// TIA Portal project "zbiorniki" (V15)

(* hardware
DEVICE "S7-1200 station_1"  S7-1200 Station
   slot 0: "Rack_0"  S7-1200 Rack  Rack  V1.0
   slot 1: "PLC_1"  CPU 1214C DC/DC/DC  6ES7 214-1AG40-0XB0  V4.2
      slot 3: "AQ 1x12BIT_1"  AQ1 signal board  6ES7 232-4HA30-0XB0  V1.0
   slot 101: "CM 1243-5"  CM 1243-5  6GK7 243-5DX30-0XE0  V1.3
   slot 102: "CM 1241 (RS485)_1"  CM 1241 (RS485)  6ES7 241-1CH30-0XB0  V1.0
*)

// ===== PLC "PLC_1"  CPU 1214C DC/DC/DC =====

VAR_GLOBAL   // PLC tag table "Default tag table"
   "czujnikDol1" AT %I0.0 : Bool;
   "czujnikGora1" AT %I0.1 : Bool;
   "Tag_2" AT %M0.0 : Bool;
   "Tag_3" AT %M0.1 : Bool;
   "Tag_4" AT %M0.2 : Bool;
   "Tag_5" AT %M2.0 : Bool;
   "poziomWodyZbiornik2" AT %MW1 : Int;
   "Tag_6" AT %IW64 : Int;
   "analog" AT %MD100 : Real;
   "skalowana" AT %MW104 : Int;
   "czujnikD2" AT %I0.2 : Bool;
   "czujnikG2" AT %I0.3 : Bool;
   "Tag_9" AT %M50.0 : Bool;
   "Tag_10" AT %M50.1 : Bool;
   "Tag_11" AT %M50.2 : Bool;
END_VAR

DATA_BLOCK "zbiornik_DB1"   // DB1
{ S7_Optimized_Access := 'TRUE' }
VERSION : 0.1
// stored: InstanceOfName zbiornik
"zbiornik"
BEGIN
   poziomCieczy := 1000;
END_DATA_BLOCK

DATA_BLOCK "pompa_DB1"   // DB2
{ S7_Optimized_Access := 'TRUE' }
VERSION : 0.1
// stored: InstanceOfName pompa
"pompa"
BEGIN
END_DATA_BLOCK

DATA_BLOCK "zbiornik_DB2"   // DB3
{ S7_Optimized_Access := 'TRUE' }
VERSION : 0.1
// stored: InstanceOfName zbiornik
"zbiornik"
BEGIN
   poziomCieczy := 500;
END_DATA_BLOCK

DATA_BLOCK "pompa_DB2"   // DB4
{ S7_Optimized_Access := 'TRUE' }
VERSION : 0.1
// stored: InstanceOfName pompa
"pompa"
BEGIN
END_DATA_BLOCK

FUNCTION_BLOCK "zbiornik"   // FB1, LAD
{ S7_Optimized_Access := 'TRUE' }
VERSION : 0.1
   VAR_INPUT
      czujnikD : Bool;
      czujnikG : Bool;
   END_VAR
   VAR_OUTPUT
      zbiornikPusty : Bool;
      zbiornikPolowa : Bool;
      zbiornikPelen : Bool;
   END_VAR
   VAR_IN_OUT
      poziomCieczy : Int;
   END_VAR
BEGIN

REGION Network 1: zbiornik pusty
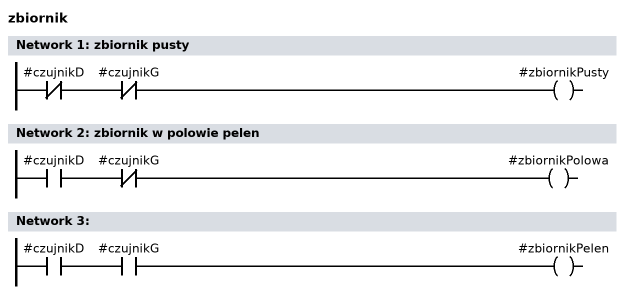
   RUNG wire#powerrail
      I_Contact( #czujnikD )
      I_Contact( #czujnikG )
      Coil( #zbiornikPusty )
   END_RUNG
   // the same network as SCL:
   #zbiornikPusty := NOT #czujnikD AND NOT #czujnikG;
END_REGION

REGION Network 2: zbiornik w polowie pelen
   RUNG wire#powerrail
      Contact( #czujnikD )
      I_Contact( #czujnikG )
      Coil( #zbiornikPolowa )
   END_RUNG
   // the same network as SCL:
   #zbiornikPolowa := #czujnikD AND NOT #czujnikG;
END_REGION

REGION Network 3
   RUNG wire#powerrail
      Contact( #czujnikD )
      Contact( #czujnikG )
      Coil( #zbiornikPelen )
   END_RUNG
   // the same network as SCL:
   #zbiornikPelen := #czujnikD AND #czujnikG;
END_REGION
END_FUNCTION_BLOCK

FUNCTION_BLOCK "pompa"   // FB2, LAD
{ S7_Optimized_Access := 'TRUE' }
VERSION : 0.1
   VAR_INPUT
      poziomCieczy : Int;
      poziomGorny : Bool;
      wysokosc : Int;
   END_VAR
   VAR_IN_OUT
      pracaPompyZb1 : Bool;
   END_VAR
BEGIN

REGION Network 1: praca pompy
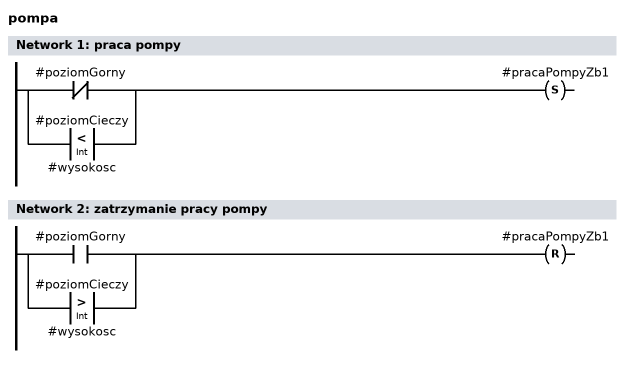
   RUNG wire#powerrail
      I_Contact( #poziomGorny )
      wire#w1
      S_Coil( #pracaPompyZb1 )
   END_RUNG
   RUNG wire#powerrail
      { S7_Templates := "SrcType := Int" } LT_Contact(in1 := #poziomCieczy, in2 := #wysokosc)
   END_RUNG wire#w1
   // the same network as SCL:
   IF NOT #poziomGorny OR (#poziomCieczy < #wysokosc) THEN #pracaPompyZb1 := TRUE; END_IF;
END_REGION

REGION Network 2: zatrzymanie pracy pompy
   RUNG wire#powerrail
      Contact( #poziomGorny )
      wire#w1
      R_Coil( #pracaPompyZb1 )
   END_RUNG
   RUNG wire#powerrail
      { S7_Templates := "SrcType := Int" } GT_Contact(in1 := #poziomCieczy, in2 := #wysokosc)
   END_RUNG wire#w1
   // the same network as SCL:
   IF #poziomGorny OR (#poziomCieczy > #wysokosc) THEN #pracaPompyZb1 := FALSE; END_IF;
END_REGION
END_FUNCTION_BLOCK

FUNCTION "przeplyw" : Void   // FC1, LAD
{ S7_Optimized_Access := 'TRUE' }
VERSION : 0.1
   VAR_INPUT
      zbiornik1 : Int;
      zmiana : Int;
      zbiornik2 : Int;
   END_VAR
   VAR_OUTPUT
      roznicaZbiornk1 : Int;
      roznicaZbiornik2 : Int;
   END_VAR
BEGIN

REGION Network 1: poziom wody w zbiorniku 2
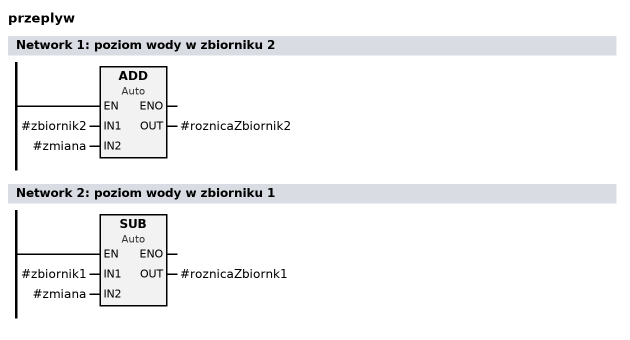
   RUNG wire#powerrail
      Add(in1 := #zbiornik2, in2 := #zmiana, out => #roznicaZbiornik2)
   END_RUNG
   // the same network as SCL:
   #roznicaZbiornik2 := #zbiornik2 + #zmiana;
END_REGION

REGION Network 2: poziom wody w zbiorniku 1
   RUNG wire#powerrail
      Sub(in1 := #zbiornik1, in2 := #zmiana, out => #roznicaZbiornk1)
   END_RUNG
   // the same network as SCL:
   #roznicaZbiornk1 := #zbiornik1 - #zmiana;
END_REGION
END_FUNCTION

ORGANIZATION_BLOCK "Main"   // OB1, LAD, ProgramCycle
TITLE = "Main Program Sweep (Cycle)"
{ S7_Optimized_Access := 'TRUE' }
VERSION : 0.1
   VAR_INPUT
      Initial_Call : Bool;   // Initial call of this OB
      Remanence : Bool;   // =True, if remanent data are available
   END_VAR
BEGIN

REGION Network 1: odczyt analogowy (poziom cieczy)
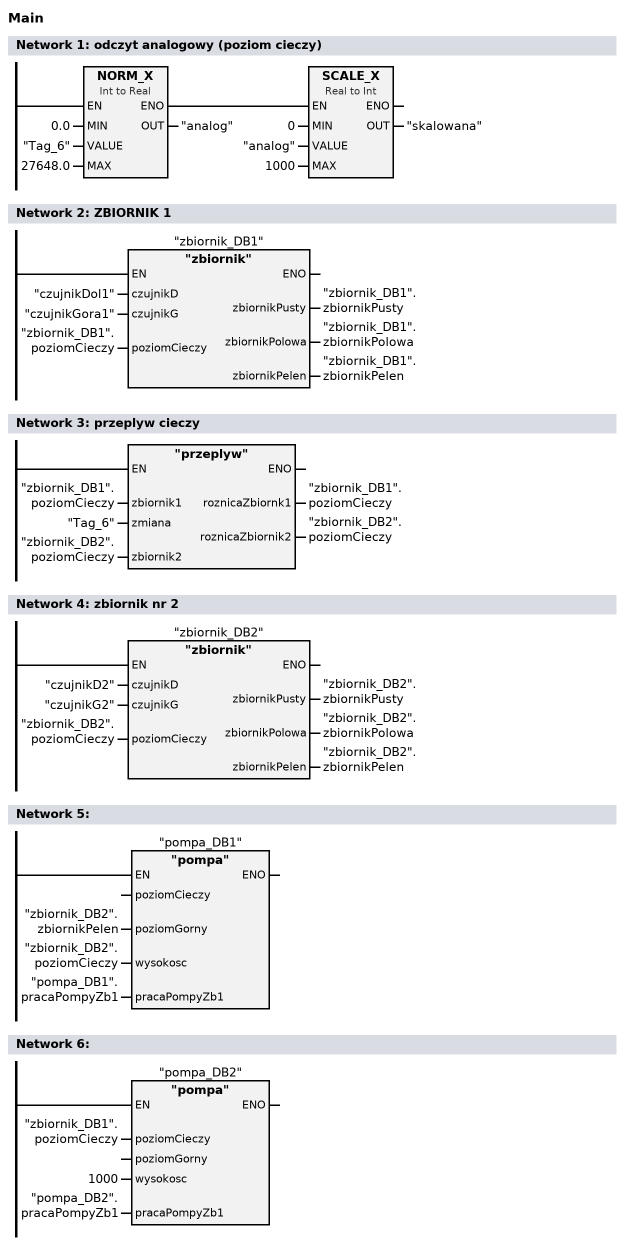
   RUNG wire#powerrail
      { S7_Templates := "[SrcType := Int, DestType := Real]" } Normalize(min := 0.0, value := "Tag_6", max := 27648.0, out => "analog")
      { S7_Templates := "[SrcType := Real, DestType := Int]" } Scale(min := 0, value := "analog", max := 1000, out => "skalowana")
   END_RUNG
   // the same network as SCL:
   "analog" := NORM_X(MIN := 0.0, VALUE := "Tag_6", MAX := 27648.0);
   "skalowana" := SCALE_X(MIN := 0, VALUE := "analog", MAX := 1000);
END_REGION

REGION Network 2: ZBIORNIK 1
   RUNG wire#powerrail
      "zbiornik_DB1"(czujnikD := "czujnikDol1", czujnikG := "czujnikGora1", poziomCieczy := "zbiornik_DB1".poziomCieczy, zbiornikPusty => "zbiornik_DB1".zbiornikPusty, zbiornikPolowa => "zbiornik_DB1".zbiornikPolowa, zbiornikPelen => "zbiornik_DB1".zbiornikPelen)
   END_RUNG
   // the same network as SCL:
   "zbiornik_DB1"(czujnikD := "czujnikDol1",   // "zbiornik"
                  czujnikG := "czujnikGora1",
                  poziomCieczy := "zbiornik_DB1".poziomCieczy,
                  zbiornikPusty => "zbiornik_DB1".zbiornikPusty,
                  zbiornikPolowa => "zbiornik_DB1".zbiornikPolowa,
                  zbiornikPelen => "zbiornik_DB1".zbiornikPelen);
END_REGION

REGION Network 3: przeplyw cieczy
   RUNG wire#powerrail
      "przeplyw"(zbiornik1 := "zbiornik_DB1".poziomCieczy, zmiana := "Tag_6", zbiornik2 := "zbiornik_DB2".poziomCieczy, roznicaZbiornk1 => "zbiornik_DB1".poziomCieczy, roznicaZbiornik2 => "zbiornik_DB2".poziomCieczy)
   END_RUNG
   // the same network as SCL:
   "przeplyw"(zbiornik1 := "zbiornik_DB1".poziomCieczy,
              zmiana := "Tag_6",
              zbiornik2 := "zbiornik_DB2".poziomCieczy,
              roznicaZbiornk1 => "zbiornik_DB1".poziomCieczy,
              roznicaZbiornik2 => "zbiornik_DB2".poziomCieczy);
END_REGION

REGION Network 4: zbiornik nr 2
   RUNG wire#powerrail
      "zbiornik_DB2"(czujnikD := "czujnikD2", czujnikG := "czujnikG2", poziomCieczy := "zbiornik_DB2".poziomCieczy, zbiornikPusty => "zbiornik_DB2".zbiornikPusty, zbiornikPolowa => "zbiornik_DB2".zbiornikPolowa, zbiornikPelen => "zbiornik_DB2".zbiornikPelen)
   END_RUNG
   // the same network as SCL:
   "zbiornik_DB2"(czujnikD := "czujnikD2",   // "zbiornik"
                  czujnikG := "czujnikG2",
                  poziomCieczy := "zbiornik_DB2".poziomCieczy,
                  zbiornikPusty => "zbiornik_DB2".zbiornikPusty,
                  zbiornikPolowa => "zbiornik_DB2".zbiornikPolowa,
                  zbiornikPelen => "zbiornik_DB2".zbiornikPelen);
END_REGION

REGION Network 5
   RUNG wire#powerrail
      "pompa_DB1"(poziomCieczy :=, poziomGorny := "zbiornik_DB2".zbiornikPelen, wysokosc := "zbiornik_DB2".poziomCieczy, pracaPompyZb1 := "pompa_DB1".pracaPompyZb1)
   END_RUNG
   // the same network as SCL:
   "pompa_DB1"(poziomGorny := "zbiornik_DB2".zbiornikPelen,   // "pompa"
               wysokosc := "zbiornik_DB2".poziomCieczy,
               pracaPompyZb1 := "pompa_DB1".pracaPompyZb1);
END_REGION

REGION Network 6
   RUNG wire#powerrail
      "pompa_DB2"(poziomCieczy := "zbiornik_DB1".poziomCieczy, poziomGorny :=, wysokosc := 1000, pracaPompyZb1 := "pompa_DB2".pracaPompyZb1)
   END_RUNG
   // the same network as SCL:
   "pompa_DB2"(poziomCieczy := "zbiornik_DB1".poziomCieczy,   // "pompa"
               wysokosc := 1000,
               pracaPompyZb1 := "pompa_DB2".pracaPompyZb1);
END_REGION
END_ORGANIZATION_BLOCK